METHOD PUBLIC ForceSafe : E_RpcMethodResponse
VAR_INPUT
    eRequester : E_Requester := E_Requester.PROG;
END_VAR
// Reject invalid identity before any command-specific mutation.
ForceSafe := F_ValidateRequester(eRequester := eRequester, bSourceLocked := FALSE, bFaulted := FALSE);
IF ForceSafe <> E_RpcMethodResponse.ACCEPTED THEN RETURN; END_IF;
_SyncConfiguration();
_operatorMailbox.CancelNormal();
_safeRequested := TRUE;
_armed := FALSE;
_forceSafe := TRUE;
_requestSync := 0.0;
_savedCommand := _requestSync;
_savedCommandValid := FALSE;
_AcceptCommand(eRequester := eRequester);
ForceSafe := E_RpcMethodResponse.ACCEPTED;
END_METHOD

{attribute 'TcRpcEnable' := '1'}
METHOD PUBLIC OperatorForceSafe : E_RpcMethodResponse
VAR_INPUT requestId : ULINT; END_VAR
OperatorForceSafe := _operatorMailbox.Submit(requestId := requestId, command := E_OperatorCommand.ForceSafe, value := 0.0);
END_METHOD

METHOD PUBLIC Reset : E_RpcMethodResponse
VAR_INPUT
    eRequester : E_Requester := E_Requester.PROG;
END_VAR
// Reject invalid identity before any command-specific mutation.
Reset := F_ValidateRequester(eRequester := eRequester, bSourceLocked := FALSE, bFaulted := FALSE);
IF Reset <> E_RpcMethodResponse.ACCEPTED THEN RETURN; END_IF;
_SyncConfiguration();
_operatorMailbox.CancelNormal();
ForceSafe(eRequester := eRequester);
Reset := SUPER^.Reset(eRequester := eRequester);
END_METHOD

METHOD PROTECTED _DispatchOperatorCommand : E_RpcMethodResponse
VAR_INPUT command : E_OperatorCommand; value : REAL; END_VAR
CASE command OF
E_OperatorCommand.SetValue: _DispatchOperatorCommand := THIS^.SetValue(rValue := value, eRequester := E_Requester.OPERATOR);
E_OperatorCommand.ForceSafe: _DispatchOperatorCommand := THIS^.ForceSafe(eRequester := E_Requester.OPERATOR);
ELSE _DispatchOperatorCommand := SUPER^._DispatchOperatorCommand(command := command, value := value);
END_CASE;
END_METHOD

METHOD PRIVATE _SyncConfiguration
VAR changed : BOOL; END_VAR
// Configuration is owned by the same cyclic task as this device.
// The first observation establishes a baseline and preserves first-scan commands.
IF NOT _configurationKnown THEN
    _lastConfiguration := cfg;
    _configurationKnown := TRUE;
    RETURN;
END_IF;
// Classify both snapshots: invalid-to-valid recovery still has invalid previous bits.
changed := NOT (F_IsFiniteReal(cfg.safeRaw) AND
    F_IsFiniteReal(cfg.euMin) AND
    F_IsFiniteReal(cfg.euMax) AND
    F_IsFiniteReal(cfg.rawMin) AND
    F_IsFiniteReal(cfg.rawMax) AND
    F_IsFiniteReal(cfg.minCv) AND
    F_IsFiniteReal(cfg.maxCv) AND
    F_IsFiniteReal(_lastConfiguration.safeRaw) AND
    F_IsFiniteReal(_lastConfiguration.euMin) AND
    F_IsFiniteReal(_lastConfiguration.euMax) AND
    F_IsFiniteReal(_lastConfiguration.rawMin) AND
    F_IsFiniteReal(_lastConfiguration.rawMax) AND
    F_IsFiniteReal(_lastConfiguration.minCv) AND
    F_IsFiniteReal(_lastConfiguration.maxCv));
IF NOT changed THEN
    changed := cfg.restoreCommandOnRestart <> _lastConfiguration.restoreCommandOnRestart OR
   cfg.holdOnBadQuality <> _lastConfiguration.holdOnBadQuality OR
   cfg.safeRaw <> _lastConfiguration.safeRaw OR
   cfg.outputType <> _lastConfiguration.outputType OR
   cfg.useRawValue <> _lastConfiguration.useRawValue OR
   cfg.minCv <> _lastConfiguration.minCv OR
   cfg.maxCv <> _lastConfiguration.maxCv OR
   cfg.euMin <> _lastConfiguration.euMin OR
   cfg.euMax <> _lastConfiguration.euMax OR
   cfg.rawMin <> _lastConfiguration.rawMin OR
   cfg.rawMax <> _lastConfiguration.rawMax OR
   cfg.clampAsFault <> _lastConfiguration.clampAsFault OR
   cfg.qualityFaultAfter <> _lastConfiguration.qualityFaultAfter;
END_IF;
IF changed THEN
    // Discard old operating intent before interpreting it under a new configuration.
    _operatorMailbox.CancelNormal();
    _armed := FALSE;
    _forceSafe := TRUE;
    _requestSync := 0.0;
    _savedCommand := 0.0;
    _savedCommandValid := FALSE;
    _commandReceived := TRUE;
    _tonBadQuality(IN := FALSE);
END_IF;
_lastConfiguration := cfg;
END_METHOD

// Runtime provenance gate, overridable by policy-test probes without system writes.
// A successful load does not establish that the latest command was durably saved.
METHOD PROTECTED _HasTrustedPersistentImage : BOOL
_HasTrustedPersistentImage := TwinCAT_SystemInfoVarList._AppInfo.BootDataLoaded
    AND NOT TwinCAT_SystemInfoVarList._AppInfo.OldBootData;
END_METHOD

END_FUNCTION_BLOCK

// ---- POUs/Alarms/Common/FB_AlarmBase.TcPOU
// Abstract base for every FB_Alarm*. Owns the common moving parts:
//   - debounce (TON/TOF) driven by cfg.common.tOnDelay / tOffDelay
//   - latch / ack bookkeeping (VAR PERSISTENT; restoration depends on the
//     application's configured and verified persistent-data saving mechanism)
//   - rising / falling / ack timestamps (LTIME)
//   - program Ack / LockSource methods and queued OperatorAck RPC
//   - the shared ST_Alarm_Sts status surface
//
// Concrete alarms:
//   - EXTEND this FB
//   - declare their own cfg : ST_Alarm<Type>_Cfg (with a nested `common : ST_Alarm_Cfg`)
//     plus any extra signal inputs
//   - compute a raw boolean trip condition from cfg + inputs
//   - call _Evaluate(cfgCommon := cfg.common, bRawCondition := ...) ONCE per
//     cycle from their body
//
// The base deliberately keeps a very small API surface — children should
// never write into sts, the timers, or the latch flags directly.
{attribute 'OPC.UA.DA' := '1'}
FUNCTION_BLOCK ABSTRACT FB_AlarmBase IMPLEMENTS I_Alarm
VAR_OUTPUT
    {attribute 'OPC.UA.DA' := '1'}
    {attribute 'OPC.UA.DA.Access' := '1'}
    sts : ST_Alarm_Sts;
END_VAR
VAR
    {attribute 'OPC.UA.DA' := '0'}
    {attribute 'OPC.UA.DA' := '0'}
    _operatorMailbox : FB_OperatorMailbox;
    {attribute 'OPC.UA.DA' := '0'}
    bSourceLockedToProg : BOOL;
    {attribute 'OPC.UA.DA' := '0'}
    _ton : TON;
    {attribute 'OPC.UA.DA' := '0'}
    _tof : TON;
    {attribute 'OPC.UA.DA' := '0'}
    _prevDebounced : BOOL;
    _commonKnown : BOOL;
    _previousCommon : ST_Alarm_Cfg;
END_VAR
VAR PERSISTENT
    // A restored latch preserves its acknowledgment state. Restart does not
    // require a second Ack; a restored acknowledged latch still needs valid
    // clear evidence. Persistent-image durability is an application concern.
    _latchedSync : BOOL;
    _ackedSync   : BOOL;
END_VAR

// Abstract base — children provide the cyclic body and call _Evaluate().

METHOD PROTECTED _DispatchOperatorCommand : E_RpcMethodResponse
VAR_INPUT command : E_OperatorCommand; value : REAL; END_VAR
CASE command OF
E_OperatorCommand.Ack: _DispatchOperatorCommand := THIS^.Ack(eRequester := E_Requester.OPERATOR);
ELSE _DispatchOperatorCommand := E_RpcMethodResponse.REJECTED_INVALID_PARAMETER;
END_CASE;
END_METHOD

// Called once per cycle by the concrete child. Takes the child's flattened
// common cfg and the pre-computed raw trip condition, and does the rest:
// debounce → latch/ack → severity → timestamps → sts.
METHOD PROTECTED _Evaluate
VAR_INPUT
    cfgCommon     : ST_Alarm_Cfg;
    bRawCondition : BOOL;
    evaluation : E_AlarmEvaluation := E_AlarmEvaluation.Valid;
    resetTiming : BOOL := FALSE;
END_VAR
VAR changed, severityValid : BOOL; END_VAR
_ProcessOperatorCommands();
sts.enabled := cfgCommon.bEnable;
sts.sMessage := cfgCommon.sMessage;
sts.evaluationState := evaluation;
// Explicit disable remains a deliberate suppression/clear operation.
IF NOT cfgCommon.bEnable THEN
    _ton(IN := FALSE); _tof(IN := FALSE);
    _latchedSync := FALSE; _ackedSync := FALSE; _prevDebounced := FALSE;
    sts.raw := FALSE; sts.debounced := FALSE; sts.active := FALSE;
    sts.latched := FALSE; sts.acked := FALSE; sts.eSeverity := E_AlarmSeverity.NONE;
    sts.valid := FALSE; sts.evaluationState := E_AlarmEvaluation.Disabled;
    _previousCommon := cfgCommon; _commonKnown := TRUE;
    RETURN;
END_IF;
// NONE is a legitimate configured severity; reject only unknown enum values.
severityValid := cfgCommon.eSeverity = E_AlarmSeverity.NONE OR cfgCommon.eSeverity = E_AlarmSeverity.INFO OR
    cfgCommon.eSeverity = E_AlarmSeverity.WARNING OR cfgCommon.eSeverity = E_AlarmSeverity.CRITICAL OR
    cfgCommon.eSeverity = E_AlarmSeverity.SHUTDOWN;
IF NOT severityValid THEN
    sts.evaluationState := E_AlarmEvaluation.InvalidConfig;
END_IF;
// A restored latch has no volatile status history yet. Publish its configured
// severity before an invalid-input return; later invalid scans preserve it.
IF NOT _commonKnown AND _latchedSync AND severityValid THEN
    sts.eSeverity := cfgCommon.eSeverity;
END_IF;
changed := _commonKnown AND (cfgCommon.tOnDelay <> _previousCommon.tOnDelay OR
    cfgCommon.tOffDelay <> _previousCommon.tOffDelay OR cfgCommon.bRequireAck <> _previousCommon.bRequireAck);
_previousCommon := cfgCommon; _commonKnown := TRUE;
IF changed OR resetTiming THEN _ton(IN := FALSE); _tof(IN := FALSE); END_IF;
sts.valid := sts.evaluationState = E_AlarmEvaluation.Valid;
IF NOT sts.valid THEN
    // Unknown evidence cannot clear an existing alarm or count toward debounce.
    _ton(IN := FALSE); _tof(IN := FALSE);
    sts.raw := FALSE;
    sts.active := sts.active OR _latchedSync;
    sts.latched := _latchedSync AND NOT _ackedSync;
    sts.acked := _ackedSync;
    RETURN;
END_IF;
sts.raw := bRawCondition;
// Debounce each state transition separately. A held active condition cannot
// disappear merely because its trip timer was reset while evidence was invalid.
IF bRawCondition THEN
    _tof(IN := FALSE);
    IF NOT sts.debounced THEN
        _ton(IN := TRUE, PT := cfgCommon.tOnDelay);
        IF _ton.Q THEN sts.debounced := TRUE; END_IF;
    ELSE _ton(IN := FALSE); END_IF;
ELSE
    _ton(IN := FALSE);
    IF sts.debounced THEN
        _tof(IN := TRUE, PT := cfgCommon.tOffDelay);
        IF _tof.Q THEN sts.debounced := FALSE; END_IF;
    ELSE _tof(IN := FALSE); END_IF;
END_IF;
IF sts.debounced AND NOT _prevDebounced THEN sts.tsTripped := F_Now();
ELSIF NOT sts.debounced AND _prevDebounced THEN sts.tsCleared := F_Now(); END_IF;
_prevDebounced := sts.debounced;
IF cfgCommon.bRequireAck AND sts.debounced AND NOT _latchedSync THEN
    _latchedSync := TRUE; _ackedSync := FALSE;
END_IF;
// Existing latches outlive changes to the policy for future trips.
IF _latchedSync AND _ackedSync AND NOT sts.debounced THEN
    _latchedSync := FALSE; _ackedSync := FALSE;
END_IF;
sts.active := sts.debounced OR _latchedSync;
sts.latched := _latchedSync AND NOT _ackedSync;
sts.acked := _ackedSync;
IF sts.active THEN sts.eSeverity := cfgCommon.eSeverity;
ELSE sts.eSeverity := E_AlarmSeverity.NONE; END_IF;
END_METHOD

METHOD PROTECTED _ProcessOperatorCommands
VAR command : E_OperatorCommand; value : REAL; result : E_RpcMethodResponse; END_VAR
IF _operatorMailbox.BeginConsume(command => command, value => value) THEN
    result := THIS^._DispatchOperatorCommand(command := command, value := value);
    _operatorMailbox.EndConsume(result := result);
END_IF;
END_METHOD

// Acknowledge the current latch. Idempotent — repeated Acks on the same latch
// just refresh tsAcked / ackRequester. If the condition has already cleared,
// the next cyclic _Evaluate releases the latch.
METHOD PUBLIC Ack : E_RpcMethodResponse
VAR_INPUT
    eRequester : E_Requester := E_Requester.PROG;
END_VAR
// Reject invalid identity before any command-specific mutation.
Ack := F_ValidateRequester(eRequester := eRequester, bSourceLocked := FALSE, bFaulted := FALSE);
IF Ack <> E_RpcMethodResponse.ACCEPTED THEN RETURN; END_IF;
Ack := F_ValidateRequester(
    eRequester    := eRequester,
    bSourceLocked := bSourceLockedToProg,
    bFaulted      := FALSE);

IF Ack = E_RpcMethodResponse.ACCEPTED AND _latchedSync THEN
    _ackedSync        := TRUE;
    sts.ackRequester  := eRequester;
    sts.tsAcked       := F_Now();
END_IF;
END_METHOD

// When bLock = TRUE, only PROG requesters may Ack(); OPERATOR calls are
// rejected with REJECTED_SOURCE_NOT_ALLOWED. Use for interlock-grade alarms
// that must only be cleared by sequence logic.
METHOD PUBLIC LockSource : E_RpcMethodResponse
VAR_INPUT
    bLock : BOOL;
END_VAR
bSourceLockedToProg := bLock;
LockSource := E_RpcMethodResponse.ACCEPTED;
END_METHOD

{attribute 'TcRpcEnable' := '1'}
METHOD PUBLIC OperatorAck : E_RpcMethodResponse

VAR_INPUT requestId : ULINT; END_VAR
OperatorAck := _operatorMailbox.Submit(requestId := requestId, command := E_OperatorCommand.Ack, value := 0.0);
END_METHOD

{attribute 'TcRpcEnable' := '1'}
METHOD PUBLIC OperatorCommandResult : E_RpcMethodResponse
VAR_INPUT requestId : ULINT; END_VAR
OperatorCommandResult := _operatorMailbox.GetResult(requestId := requestId);
END_METHOD

METHOD PROTECTED _InvalidateEvaluation
VAR_INPUT evaluation : E_AlarmEvaluation; END_VAR
_ton(IN := FALSE); _tof(IN := FALSE);
sts.valid := FALSE; sts.evaluationState := evaluation; sts.raw := FALSE;
// Preserve established alarm state and timestamps until fresh valid evidence.
END_METHOD

END_FUNCTION_BLOCK

// ---- POUs/Alarms/Simple/FB_AlarmSimple.TcPOU
// Debounced / latchable boolean mirror. Use to wrap any digital condition the
// HMI should see through the standard alarm surface (severity, ack,
// timestamps, message) — e.g. a device-fault rollup, a door-open switch, an
// e-stop echo, or a plant-level boolean computed elsewhere.
//
// Usage:
//   almDoorOpen.cfg.common.bEnable   := TRUE;
//   almDoorOpen.cfg.common.eSeverity := E_AlarmSeverity.WARNING;
//   almDoorOpen.cfg.common.tOnDelay  := T#2S;
//   almDoorOpen.cfg.common.sMessage  := 'Cell door open';
//   almDoorOpen(inpActive := GVL_HW.DOOR_SW.sts.value);
{attribute 'OPC.UA.DA' := '1'}
FUNCTION_BLOCK FB_AlarmSimple EXTENDS FB_AlarmBase
VAR_INPUT
    // Application quality gate; FALSE means no trustworthy new evidence.
    inpValid : BOOL := TRUE;
    {attribute 'OPC.UA.DA' := '1'}
    {attribute 'OPC.UA.DA.Access' := '1'}
    cfg       : ST_AlarmSimple_Cfg;

    {attribute 'OPC.UA.DA' := '0'}
    inpActive : BOOL;
END_VAR

IF inpValid THEN
    _Evaluate(cfgCommon := cfg.common, bRawCondition := inpActive);
ELSE
    _Evaluate(cfgCommon := cfg.common, bRawCondition := FALSE, evaluation := E_AlarmEvaluation.InvalidInput);
END_IF;

END_FUNCTION_BLOCK

// ---- POUs/Alarms/Threshold/FB_AlarmThreshold.TcPOU
// Single-direction threshold alarm over a REAL process value.
//
// Usage (high temp warning with 2s debounce, latching + ack):
//   almHi.cfg.common.bEnable     := TRUE;
//   almHi.cfg.common.tOnDelay    := T#2S;
//   almHi.cfg.common.bRequireAck := TRUE;
//   almHi.cfg.common.eSeverity   := E_AlarmSeverity.WARNING;
//   almHi.cfg.common.sMessage    := 'Reactor T > 80C';
//   almHi.cfg.fThreshold         := 80.0;
//   almHi.cfg.bFailHigh          := TRUE;
//   almHi(inpValue := reactorTempC);
{attribute 'OPC.UA.DA' := '1'}
FUNCTION_BLOCK FB_AlarmThreshold EXTENDS FB_AlarmBase
VAR_INPUT
    // Application quality gate; FALSE means no trustworthy new evidence.
    inpValid : BOOL := TRUE;
    {attribute 'OPC.UA.DA' := '1'}
    {attribute 'OPC.UA.DA.Access' := '1'}
    cfg      : ST_AlarmThreshold_Cfg;

    {attribute 'OPC.UA.DA' := '0'}
    inpValue : REAL;
END_VAR
VAR
    _criteriaKnown : BOOL;
    _criteriaChanged : BOOL;
    _previousCriteria : ST_AlarmThreshold_Cfg;
    _evaluation : E_AlarmEvaluation;
    {attribute 'OPC.UA.DA' := '0'}
    _raw : BOOL;
END_VAR

_criteriaChanged := FALSE;
IF _criteriaKnown THEN
    IF NOT (F_IsFiniteReal(cfg.fThreshold) AND F_IsFiniteReal(_previousCriteria.fThreshold)) THEN _criteriaChanged := TRUE;
    ELSE _criteriaChanged := cfg.fThreshold <> _previousCriteria.fThreshold OR cfg.bFailHigh <> _previousCriteria.bFailHigh OR cfg.bFailLow <> _previousCriteria.bFailLow; END_IF;
END_IF;
_criteriaKnown := TRUE; _previousCriteria := cfg;
_raw := FALSE;
_evaluation := E_AlarmEvaluation.Valid;
IF NOT F_IsFiniteReal(cfg.fThreshold) OR (cfg.bFailHigh = cfg.bFailLow) THEN
    _evaluation := E_AlarmEvaluation.InvalidConfig;
ELSIF NOT inpValid OR NOT F_IsFiniteReal(inpValue) THEN
    _evaluation := E_AlarmEvaluation.InvalidInput;
ELSIF cfg.bFailHigh THEN _raw := inpValue > cfg.fThreshold;
ELSE _raw := inpValue < cfg.fThreshold;
END_IF;
_Evaluate(cfgCommon := cfg.common, bRawCondition := _raw, evaluation := _evaluation, resetTiming := _criteriaChanged);

END_FUNCTION_BLOCK

// ---- POUs/Alarms/Limit/FB_AlarmLimit.TcPOU
// Four-level limit ladder (HiHi / Hi / Lo / LoLo) built on four composed
// FB_AlarmThreshold instances. Each level has its own full config; delays,
// severity, and ack behaviour are set per level.
//
// Flood suppression: HiHi hides Hi, LoLo hides Lo on the rollup flags. The
// raw sub-statuses (HiHi / Hi / Lo / LoLo) are still exposed for forensics.
//
// Ack() cascades to every sub-alarm. LockSource() cascades identically, so the
// composite honours a single source-lock decision.
//
// Typical config (alongside an analog input):
//   cfg.HiHi.common.bEnable := TRUE; cfg.HiHi.fThreshold := 110.0;
//   cfg.HiHi.bFailHigh := TRUE;      cfg.HiHi.common.eSeverity := E_AlarmSeverity.CRITICAL;
//   cfg.Hi.common.bEnable   := TRUE; cfg.Hi.fThreshold   := 100.0;
//   cfg.Hi.bFailHigh   := TRUE;      cfg.Hi.common.eSeverity   := E_AlarmSeverity.WARNING;
//   cfg.Lo.common.bEnable   := TRUE; cfg.Lo.fThreshold   :=  20.0;
//   cfg.Lo.bFailLow    := TRUE;      cfg.Lo.common.eSeverity   := E_AlarmSeverity.WARNING;
//   cfg.LoLo.common.bEnable := TRUE; cfg.LoLo.fThreshold :=  10.0;
//   cfg.LoLo.bFailLow  := TRUE;      cfg.LoLo.common.eSeverity := E_AlarmSeverity.CRITICAL;
{attribute 'OPC.UA.DA' := '1'}
FUNCTION_BLOCK FB_AlarmLimit IMPLEMENTS I_Alarm
VAR_INPUT
    // Application quality gate; FALSE means no trustworthy new evidence.
    inpValid : BOOL := TRUE;
    {attribute 'OPC.UA.DA' := '1'}
    {attribute 'OPC.UA.DA.Access' := '1'}
    cfg   : ST_AlarmLimit_Cfg;

    {attribute 'OPC.UA.DA' := '0'}
    inpPv : REAL;
END_VAR
VAR_OUTPUT
    {attribute 'OPC.UA.DA' := '1'}
    {attribute 'OPC.UA.DA.Access' := '1'}
    sts : ST_AlarmLimit_Sts;
END_VAR
VAR
    {attribute 'OPC.UA.DA' := '0'}
    {attribute 'OPC.UA.DA' := '0'}
    _operatorMailbox : FB_OperatorMailbox;
    _hiHi : FB_AlarmThreshold;
    _hi   : FB_AlarmThreshold;
    _lo   : FB_AlarmThreshold;
    _loLo : FB_AlarmThreshold;
END_VAR

_ProcessOperatorCommands();
// Push config into each sub-alarm every cycle so HMI changes take effect.
_hiHi.cfg := cfg.HiHi;
_hi.cfg   := cfg.Hi;
_lo.cfg   := cfg.Lo;
_loLo.cfg := cfg.LoLo;

_hiHi(inpValue := inpPv, inpValid := inpValid);
_hi(inpValue   := inpPv, inpValid := inpValid);
_lo(inpValue   := inpPv, inpValid := inpValid);
_loLo(inpValue := inpPv, inpValid := inpValid);

// Expose raw sub-statuses
sts.HiHi := _hiHi.sts;
sts.Hi   := _hi.sts;
sts.Lo   := _lo.sts;
sts.LoLo := _loLo.sts;

// Disabled levels do not invalidate enabled levels; all-disabled has no evaluation.
sts.evaluationState := E_AlarmEvaluation.Disabled;
IF cfg.HiHi.common.bEnable OR cfg.Hi.common.bEnable OR cfg.Lo.common.bEnable OR cfg.LoLo.common.bEnable THEN
    sts.evaluationState := E_AlarmEvaluation.Valid;
    IF sts.HiHi.enabled AND NOT sts.HiHi.valid THEN
        IF sts.evaluationState <> E_AlarmEvaluation.InvalidConfig THEN sts.evaluationState := sts.HiHi.evaluationState; END_IF;
    END_IF;
    IF sts.Hi.enabled AND NOT sts.Hi.valid THEN
        IF sts.evaluationState <> E_AlarmEvaluation.InvalidConfig THEN sts.evaluationState := sts.Hi.evaluationState; END_IF;
    END_IF;
    IF sts.Lo.enabled AND NOT sts.Lo.valid THEN
        IF sts.evaluationState <> E_AlarmEvaluation.InvalidConfig THEN sts.evaluationState := sts.Lo.evaluationState; END_IF;
    END_IF;
    IF sts.LoLo.enabled AND NOT sts.LoLo.valid THEN
        IF sts.evaluationState <> E_AlarmEvaluation.InvalidConfig THEN sts.evaluationState := sts.LoLo.evaluationState; END_IF;
    END_IF;
END_IF;
sts.valid := sts.evaluationState = E_AlarmEvaluation.Valid;

// Rollup with suppression (higher priority hides lower on same direction)
sts.hiHiActive := _hiHi.sts.active;
sts.hiActive   := _hi.sts.active   AND NOT sts.hiHiActive;
sts.loLoActive := _loLo.sts.active;
sts.loActive   := _lo.sts.active   AND NOT sts.loLoActive;

sts.anyActive := sts.hiHiActive OR sts.hiActive OR sts.loActive OR sts.loLoActive;

// Aggregate severity — highest currently-active level wins.
sts.eSeverity := E_AlarmSeverity.NONE;
IF _hiHi.sts.eSeverity > sts.eSeverity THEN sts.eSeverity := _hiHi.sts.eSeverity; END_IF;
IF _hi.sts.eSeverity   > sts.eSeverity THEN sts.eSeverity := _hi.sts.eSeverity;   END_IF;
IF _lo.sts.eSeverity   > sts.eSeverity THEN sts.eSeverity := _lo.sts.eSeverity;   END_IF;
IF _loLo.sts.eSeverity > sts.eSeverity THEN sts.eSeverity := _loLo.sts.eSeverity; END_IF;

METHOD PROTECTED _DispatchOperatorCommand : E_RpcMethodResponse
VAR_INPUT command : E_OperatorCommand; value : REAL; END_VAR
CASE command OF
E_OperatorCommand.Ack: _DispatchOperatorCommand := THIS^.Ack(eRequester := E_Requester.OPERATOR);
ELSE _DispatchOperatorCommand := E_RpcMethodResponse.REJECTED_INVALID_PARAMETER;
END_CASE;
END_METHOD

METHOD PROTECTED _ProcessOperatorCommands
VAR command : E_OperatorCommand; value : REAL; result : E_RpcMethodResponse; END_VAR
IF _operatorMailbox.BeginConsume(command => command, value => value) THEN
    result := THIS^._DispatchOperatorCommand(command := command, value := value);
    _operatorMailbox.EndConsume(result := result);
END_IF;
END_METHOD

// Composite Ack — cascades to all four levels. Returns ACCEPTED if at least
// one level accepted; reports any source-lock rejection otherwise.
METHOD PUBLIC Ack : E_RpcMethodResponse
VAR_INPUT
    eRequester : E_Requester := E_Requester.PROG;
END_VAR
VAR
    r1, r2, r3, r4 : E_RpcMethodResponse;
END_VAR
// Reject invalid identity before any command-specific mutation.
Ack := F_ValidateRequester(eRequester := eRequester, bSourceLocked := FALSE, bFaulted := FALSE);
IF Ack <> E_RpcMethodResponse.ACCEPTED THEN RETURN; END_IF;
r1 := _hiHi.Ack(eRequester := eRequester);
r2 := _hi.Ack(eRequester   := eRequester);
r3 := _lo.Ack(eRequester   := eRequester);
r4 := _loLo.Ack(eRequester := eRequester);

IF r1 = E_RpcMethodResponse.ACCEPTED OR r2 = E_RpcMethodResponse.ACCEPTED
   OR r3 = E_RpcMethodResponse.ACCEPTED OR r4 = E_RpcMethodResponse.ACCEPTED THEN
    Ack := E_RpcMethodResponse.ACCEPTED;
ELSE
    // Every level rejected — all four reject for the same reason (source
    // lock / not latched), so returning the HiHi response is representative.
    Ack := r1;
END_IF;
END_METHOD

METHOD PUBLIC LockSource : E_RpcMethodResponse
VAR_INPUT
    bLock : BOOL;
END_VAR
_hiHi.LockSource(bLock := bLock);
_hi.LockSource(bLock   := bLock);
_lo.LockSource(bLock   := bLock);
_loLo.LockSource(bLock := bLock);
LockSource := E_RpcMethodResponse.ACCEPTED;
END_METHOD

{attribute 'TcRpcEnable' := '1'}
METHOD PUBLIC OperatorAck : E_RpcMethodResponse

VAR_INPUT requestId : ULINT; END_VAR
OperatorAck := _operatorMailbox.Submit(requestId := requestId, command := E_OperatorCommand.Ack, value := 0.0);
END_METHOD

{attribute 'TcRpcEnable' := '1'}
METHOD PUBLIC OperatorCommandResult : E_RpcMethodResponse
VAR_INPUT requestId : ULINT; END_VAR
OperatorCommandResult := _operatorMailbox.GetResult(requestId := requestId);
END_METHOD

END_FUNCTION_BLOCK

// ---- POUs/Alarms/RateOfChange/FB_AlarmRateOfChange.TcPOU
// Runaway / sensor-drop detector. Alarms when |d(inpPv)/dt| > cfg.fRateLimit.
//
// dt is measured via F_GetTaskCycleTime() so the rate is calibrated in
// engineering-units per second regardless of task rate. First scan after
// power-up or after bEnable rises initialises the previous sample and reports
// zero rate (no false trip at boot).
//
// outRateOfChange is always exposed for diagnostics / trending, not only when
// the alarm is active.
{attribute 'OPC.UA.DA' := '1'}
FUNCTION_BLOCK FB_AlarmRateOfChange EXTENDS FB_AlarmBase
VAR_INPUT
    // Application quality gate; FALSE means no trustworthy new evidence.
    inpValid : BOOL := TRUE;
    {attribute 'OPC.UA.DA' := '1'}
    {attribute 'OPC.UA.DA.Access' := '1'}
    cfg   : ST_AlarmRateOfChange_Cfg;

    {attribute 'OPC.UA.DA' := '0'}
    inpPv : REAL;
END_VAR
VAR_OUTPUT
    {attribute 'OPC.UA.DA' := '1'}
    {attribute 'OPC.UA.DA.Access' := '1'}
    {attribute 'OPC.UA.DA.Description' := 'Latest rate of change (units / s)'}
    outRateOfChange : LREAL;
END_VAR
VAR
    _evaluation : E_AlarmEvaluation;
    _task : DINT;
    _previousTask : DINT;
    _previousCycleTime : LREAL;
    _configKnown : BOOL;
    _previousLimit : REAL;
    _previousOnDelay : TIME;
    _previousOffDelay : TIME;
    _previousRequireAck : BOOL;
    {attribute 'OPC.UA.DA' := '0'}
    _raw           : BOOL;
    {attribute 'OPC.UA.DA' := '0'}
    _previousPv    : REAL;
    {attribute 'OPC.UA.DA' := '0'}
    _firstScan     : BOOL := TRUE;
    {attribute 'OPC.UA.DA' := '0'}
    _cycleTimeSec  : LREAL;
END_VAR

_raw := FALSE;
_evaluation := E_AlarmEvaluation.Valid;
_task := Tc2_System.GETCURTASKINDEXEX();
IF NOT F_IsFiniteReal(cfg.fRateLimit) THEN _evaluation := E_AlarmEvaluation.InvalidConfig;
ELSIF cfg.fRateLimit < 0.0 THEN _evaluation := E_AlarmEvaluation.InvalidConfig;
END_IF;
IF NOT (cfg.common.eSeverity = E_AlarmSeverity.NONE OR cfg.common.eSeverity = E_AlarmSeverity.INFO OR
    cfg.common.eSeverity = E_AlarmSeverity.WARNING OR cfg.common.eSeverity = E_AlarmSeverity.CRITICAL OR
    cfg.common.eSeverity = E_AlarmSeverity.SHUTDOWN) THEN _evaluation := E_AlarmEvaluation.InvalidConfig; END_IF;
IF _evaluation = E_AlarmEvaluation.Valid THEN
    IF NOT inpValid OR NOT F_IsFiniteReal(inpPv) THEN _evaluation := E_AlarmEvaluation.InvalidInput;
    END_IF;
END_IF;
IF _evaluation = E_AlarmEvaluation.Valid THEN
    IF _task <= 0 THEN _evaluation := E_AlarmEvaluation.InvalidConfig;
    ELSE
        _cycleTimeSec := TIME_TO_LREAL(F_GetTaskCycleTime()) / LREAL#1000.0;
        IF _cycleTimeSec <= 0.0 THEN _evaluation := E_AlarmEvaluation.InvalidConfig; END_IF;
    END_IF;
END_IF;
IF NOT cfg.common.bEnable OR _evaluation <> E_AlarmEvaluation.Valid THEN
    _firstScan := TRUE; _configKnown := FALSE; outRateOfChange := 0.0;
    _Evaluate(cfgCommon := cfg.common, bRawCondition := FALSE, evaluation := _evaluation);
    RETURN;
END_IF;
// Previous limit is stored only after classification; equality is now safe.
IF NOT _configKnown OR _previousTask <> _task THEN _firstScan := TRUE;
ELSIF _cycleTimeSec <> _previousCycleTime OR cfg.fRateLimit <> _previousLimit OR cfg.common.tOnDelay <> _previousOnDelay OR
    cfg.common.tOffDelay <> _previousOffDelay OR cfg.common.bRequireAck <> _previousRequireAck THEN
    _firstScan := TRUE;
END_IF;
_configKnown := TRUE; _previousLimit := cfg.fRateLimit; _previousTask := _task;
_previousCycleTime := _cycleTimeSec;
_previousOnDelay := cfg.common.tOnDelay; _previousOffDelay := cfg.common.tOffDelay;
_previousRequireAck := cfg.common.bRequireAck;
IF _firstScan THEN
    _firstScan := FALSE; _previousPv := inpPv; outRateOfChange := 0.0;
    _Evaluate(cfgCommon := cfg.common, bRawCondition := FALSE, evaluation := E_AlarmEvaluation.Initializing);
    RETURN;
END_IF;
// Widen before subtract/divide: all finite REAL extremes fit comfortably in LREAL.
outRateOfChange := (REAL_TO_LREAL(inpPv) - REAL_TO_LREAL(_previousPv)) / _cycleTimeSec;
_previousPv := inpPv;
_raw := ABS(outRateOfChange) > REAL_TO_LREAL(cfg.fRateLimit);
_Evaluate(cfgCommon := cfg.common, bRawCondition := _raw);

// Application-only owning-task API; invalidate history before assigning a new signal source.
METHOD PUBLIC ReassignInput
_firstScan := TRUE; _configKnown := FALSE; outRateOfChange := 0.0;
IF cfg.common.bEnable THEN _InvalidateEvaluation(evaluation := E_AlarmEvaluation.Initializing); END_IF;
END_METHOD

END_FUNCTION_BLOCK
